{attribute 'linkalways'} 
{attribute 'no_explicit_call' := 'This FB is a CLASS and must be accessed using methods or properties'}
{attribute 'enable_dynamic_creation'}
FUNCTION_BLOCK FINAL Node_LEN EXTENDS Node
VAR
	str : _STRING('');
	out : _INT(0);
END_VAR

METHOD PUBLIC  Clone : I_Node
VAR
	pNode : POINTER TO Node_LEN;
END_VAR
pNode := __NEW(Node_LEN);
Clone := pNode^;
END_METHOD

METHOD FB_init : BOOL
VAR_INPUT
	bInitRetains : BOOL; // if TRUE, the retain variables are initialized (warm start / cold start)
	bInCopyCode : BOOL;  // if TRUE, the instance afterwards gets moved into the copy code (online change)
END_VAR
AddParameter('str', str);
AddOutput('out', out);
END_METHOD

METHOD PROTECTED OnExecute
VAR
END_VAR
out.Value := LEN(str.Value);
END_METHOD

END_FUNCTION_BLOCK

(* stored: Version 1.1.0.1, ProductVersion 3.1.4026.18
   POU Node_LEN: Id {81fe9d1e-f9a3-0de5-0f52-55c80b5e7031}, SpecialFunc None
   Folder Constructor: Id {1734dd43-e24f-0f95-0860-c301922bb0f6}
   Method Clone: Id {f8d10471-e05c-0e6f-1b7a-53368061ebe2}
   Method FB_init: Id {922a4fa7-629d-0d21-2fda-6c7a768cdb0b}
   Method OnExecute: Id {19e5c4fd-01de-0898-2c4a-6f65db5b2d30} *)
